(* IEC 61131-3 sources: AXOpen/src/core/ctrl/src/abstractions/AxoCoordination, 2 files *)

(* ---- AxoCoordinatorStates.st ---- *)
NAMESPACE AXOpen.Core
    TYPE PUBLIC
        AxoCoordinatorStates : INT (Idle := 0, Configuring := 1, Running := 2) := Idle;
    END_TYPE
END_NAMESPACE

(* ---- IAxoCoordinator.st ---- *)
NAMESPACE AXOpen.Core
    INTERFACE  IAxoCoordinator EXTENDS IAxoObject
        METHOD GetCoordinatorState : AxoCoordinatorStates END_METHOD
        METHOD MoveNext END_METHOD
        METHOD RequestStep
            VAR_INPUT
                RequestedStep : IAxoStep;
            END_VAR
        END_METHOD
        METHOD GetCurrentStep : IAxoStep END_METHOD

    END_INTERFACE
END_NAMESPACE
